(* CODESYS project MNG_SimIO_Upd.export

Project tree, tasks and I/O mapping:
  MNG_SimIO/
    function block MNG_SIMIO_UPDATER [ST]
  data type MNG_APPLICATION_INPUTS_32BIT
  data type MNG_APPLICATION_OUTPUTS_32BIT
*)

// MNG_APPLICATION_INPUTS_32BIT
TYPE MNG_APPLICATION_INPUTS_32BIT :
STRUCT
    NumSignals                    : INT     := 10        ;
EndoflEnd_of_Line_Packaging_STEP_TriggerZaehler_out: BOOL    := 0; (* EndoflEnd_of_Line_Packaging_STEP?TriggerZaehler_out *)

Gleitschiene_Links_AXIS: REAL    := 0.0; (* ubgeruest_EndoflGreifarm_Gleitschiene_Links?KinAxis *)

Laufwagen_1_Busy: BOOL    := 0; (* _EndoflEnd_of_Line_Packaging_STEP_Laufwagen_1?Busy *)

EndoflLaufwagen_AXIS: REAL    := 0.0; (* _Packaging_STEP_Laufwagen_1_EndoflLaufwagen?KinAxis *)

EndoflLaufwagen_DLT_POS: REAL    := 0.0; (* Packaging_STEP_Laufwagen_1_EndoflLaufwagen?KinDelta *)

EndoflLaufwagen_ACT_SPD: REAL    := 0.0; (* Packaging_STEP_Laufwagen_1_EndoflLaufwagen?KinSpeed *)

EndoflLaufwagen_KinState: DINT    := 0; (* Packaging_STEP_Laufwagen_1_EndoflLaufwagen?KinState *)

EndoflLaufwagen_ZaehlerQuer: UINT    := 0; (* kaging_STEP_Laufwagen_1_EndoflLaufwagen?ZaehlerQuer *)

EndoflLaufwagen_ZaehlerLaengs: UINT    := 0; (* ging_STEP_Laufwagen_1_EndoflLaufwagen?ZaehlerLaengs *)

EndoflLaufwagen_Hubausschiebpos: REAL    := 0.0; (* ng_STEP_Laufwagen_1_EndoflLaufwagen?Hubausschiebpos *)

END_STRUCT
END_TYPE

// MNG_APPLICATION_OUTPUTS_32BIT
TYPE MNG_APPLICATION_OUTPUTS_32BIT :
STRUCT
    NumSignals                    : INT     := 6         ;
Pusher_1_Enabled: BOOL    := 0; (* _EndoflEnd_of_Line_Packaging_STEP_Pusher_1?Enabled *)

Drehschieber_Achse_1_Set_AST: BOOL    := 0; (* ng_STEP_Drehschieber_1_Drehschieber_Achse_1?Set_AST *)

Drehschieber_Achse_1_Set_GST: BOOL    := 0; (* ng_STEP_Drehschieber_1_Drehschieber_Achse_1?Set_GST *)

EndoflEnd_of_Line_Packaging_STEP_Status_out: UINT    := 0; (* _EndoflEnd_of_Line_Packaging_STEP?Status_out *)

EndoflEnd_of_Line_Packaging_STEP_Ausschieben_in: BOOL    := 0; (* _EndoflEnd_of_Line_Packaging_STEP?Ausschieben_in *)

EndoflEnd_of_Line_Packaging_STEP_Laufwagen_1_Cmd_out: UINT    := 0; (* ndoflEnd_of_Line_Packaging_STEP?Laufwagen_1_Cmd_out *)

END_STRUCT
END_TYPE

// MNG_SimIO/MNG_SIMIO_UPDATER
FUNCTION_BLOCK MNG_SIMIO_UPDATER
(* This function block implements simple TCP/IP client protocol.              *)
(* The max. size of binary tx/rx data has to be <= PLCPRJ_BUFFER_SIZE         *)
VAR_INPUT
connect : BOOL := FALSE;
IPAddress : STRING := '192.168.8.175';
port : INT := 5003;
timeout : DINT := 3;		(* Timeout in seconds *)
Q : MNG_Application_Outputs_32Bit;    (* Tx user data *)
END_VAR
VAR_OUTPUT
I      : MNG_Application_Inputs_32Bit        ; (* Rx user data *)
Counter   : DINT := 0;
Connected : BOOL := FALSE;
END_VAR
VAR
state : INT := 0;
socket : RTS_IEC_HANDLE := -1(*SOCKET_INVALID*);
bOptNoDelay: BOOL := TRUE;
sa:SOCKADDRESS;
fdRead:SOCKET_FD_SET;
tvTimeout:SOCKET_TIMEVAL;
pdiReady:DINT := 0;
toServer         : MNG_RawDatagram;
fromServer       : MNG_RawDatagram;
expectedSize, recvSize : LINT := 0;
sendSize: UDINT := 0; 
sentSize : LINT := 0;

bInit: BOOL := FALSE;
DWordBuffer      : DWORD                                               ; (* convert DWORD data *)
DIntBuffer       : DINT                                                ; (* convert DINT data *)
Segment11_F: BOOL;
Error: DINT;
diSocket: BOOL;
result: RTS_IEC_RESULT; 
callback: CB.CB_CALLBACK;
callbackError: CB.ERROR; 
END_VAR
(* @END_DECLARATION := '0'                                                    *)

IF NOT bInit THEN
//         SysCallbackRegister(INDEXOF(CallbackReset), EVENT_BEFORE_RESET);
	callback.eEvent := CB.EVENT.BEFORE_RESET;
	callback.eClass := CB.EVENT_CLASS.ALL_CLASSES;
	callback.eSource := CB.EVENT_SOURCE.ALL_SOURCES;
	callback.pPOUFunc := ADR(CallbackReset); 
	
	CB.RegisterCallback(callback, ADR(callbackError));
        bInit := TRUE;
END_IF
CASE state OF
0:											(* Init *)
  	socket := -1(*SOCKET_INVALID*);
  	Connected := FALSE;
  	IF connect THEN
  	        state  := 10;
  	END_IF
10:											(* Create socket *)
        socket := SysSockCreate(SOCKET_AF_INET, SOCKET_STREAM, 0, ADR(result));
        (*IF socket <> 0(*= SOCKET_INVALID*) THEN
            state := 100;
        ELSE
            state := 20;
        END_IF*)
		state := 20;
20:											(* Setup and Connect *)
        (* SysSockSetOption(socket, SOCKET_SOL, SOCKET_SO_SNDBUF, ADR(diMaxDataSize), SIZEOF(diMaxDataSize));
        SysSockSetOption(socket, SOCKET_SOL, SOCKET_SO_RCVBUF, ADR(diMaxDataSize), SIZEOF(diMaxDataSize));
        lOptLinger.l_onoff:=0;
        lOptLinger.l_linger:=0;
        SysSockSetOption(diSocket,	SOCKET_SOL, SOCKET_SO_LINGER, ADR(lOptLinger), SIZEOF(lOptLinger)); *)
        bOptNoDelay:=TRUE;
        SysSockSetOption(socket,	SOCKET_IPPROTO_TCP, SOCKET_TCP_NODELAY, ADR(bOptNoDelay), SIZEOF(bOptNoDelay));
        sa.sin_family:=SOCKET_AF_INET;
        sa.sin_addr.ulAddr:=GetIPAddress(IPAddress);
        tvTimeout.tv_sec := timeout ;
        tvTimeout.tv_usec := 0;
        fdRead.fd_count := 1;
        fdRead.fd_array[0] := socket;
        IF sa.sin_addr.ulAddr = SOCKET_INADDR_NONE THEN
                state := 121;
        ELSE
                 sa.sin_port:=SysSockHtons(port);
                 IF SysSockConnect(socket, ADR(sa), SIZEOF(sa)) = 0  THEN
                        state := 30;
                 ELSE
                         Error := 10035(*SysSockGetLastErrorSync(socket)*);	
						(* Query reason why connect reported failure *)
                                         CASE  Error OF
                         10035: 			(* EWOULDBLOCK *)
                                 state := 30;
                         10056: 			 (* ALREADY_CONNECTED*)
                                 state := 30;
                         ELSE
                                 state := 60;
                         END_CASE
                END_IF
        END_IF
30:											(* Data exchange *)
                Connected := TRUE;
                fdRead.fd_array[0] := socket;
                IF (SysSockSelect(SOCKET_FD_SETSIZE, ADR(fdRead), 0, 0, ADR(tvTimeout), ADR(pdiReady)) = CmpErrors.Errors.ERR_OK) AND pdiReady > 0 THEN
                expectedSize := 16 + (I.NumSignals+1) * 4;
                recvSize := SysSockRecv(socket, ADR(fromServer), expectedSize, 0, ADR(result));
                IF result <> CmpErrors.Errors.ERR_OK OR expectedSize <= 0 THEN
                         state := 60;

                ELSIF expectedSize = recvSize THEN

                        (* correct header data *)
                        fromServer.Header.ByteCount   	 := SysSockNtohl(fromServer.Header.ByteCount);
                        Counter                        				:= SysSockNtohl(fromServer.Header.Counter);
                        fromServer.Header.SentTime  	   := SysSockNtohl(fromServer.Header.SentTime);
                        fromServer.Header.DatagramType := SysSockNtohl(fromServer.Header.DatagramType);

                        (* currently only use the data on a 32 Bit raw image *)
                        IF fromServer.Header.DatagramType = MNG_DatagramType.MNG_Raw32BitImage THEN
                                                        (* BOOL EndoflEnd_of_Line_Packaging_STEP_TriggerZaehler_out *)
                                                        I.EndoflEnd_of_Line_Packaging_STEP_TriggerZaehler_out := fromServer.Payload[2] <> 0;
                                                        (* REAL Gleitschiene_Links_AXIS *)
                                                        DWordBuffer := SysSockNtohl(fromServer.Payload[3]);
                                                        SysMemCpy(pDest := ADR(I.Gleitschiene_Links_AXIS), pSrc := ADR(DWordBuffer), udiCount := 4);
                                                        (* BOOL Laufwagen_1_Busy *)
                                                        I.Laufwagen_1_Busy := fromServer.Payload[4] <> 0;
                                                        (* REAL EndoflLaufwagen_AXIS *)
                                                        DWordBuffer := SysSockNtohl(fromServer.Payload[5]);
                                                        SysMemCpy(pDest := ADR(I.EndoflLaufwagen_AXIS), pSrc := ADR(DWordBuffer), udiCount := 4);
                                                        (* REAL EndoflLaufwagen_DLT_POS *)
                                                        DWordBuffer := SysSockNtohl(fromServer.Payload[6]);
                                                        SysMemCpy(pDest := ADR(I.EndoflLaufwagen_DLT_POS), pSrc := ADR(DWordBuffer), udiCount := 4);
                                                        (* REAL EndoflLaufwagen_ACT_SPD *)
                                                        DWordBuffer := SysSockNtohl(fromServer.Payload[7]);
                                                        SysMemCpy(pDest := ADR(I.EndoflLaufwagen_ACT_SPD), pSrc := ADR(DWordBuffer), udiCount := 4);
                                                        (* DINT EndoflLaufwagen_KinState *)
                                                        DWordBuffer := SysSockNtohl(fromServer.Payload[8]);
                                                        SysMemCpy(pDest := ADR(I.EndoflLaufwagen_KinState), pSrc := ADR(DWordBuffer), udiCount := 4);
                                                        (* UINT EndoflLaufwagen_ZaehlerQuer *)
                                                        DWordBuffer := SysSockNtohl(fromServer.Payload[9]);
                                                        I.EndoflLaufwagen_ZaehlerQuer := DWORD_TO_UINT(DWordBuffer);
                                                        (* UINT EndoflLaufwagen_ZaehlerLaengs *)
                                                        DWordBuffer := SysSockNtohl(fromServer.Payload[10]);
                                                        I.EndoflLaufwagen_ZaehlerLaengs := DWORD_TO_UINT(DWordBuffer);
                                                        (* REAL EndoflLaufwagen_Hubausschiebpos *)
                                                        DWordBuffer := SysSockNtohl(fromServer.Payload[11]);
                                                        SysMemCpy(pDest := ADR(I.EndoflLaufwagen_Hubausschiebpos), pSrc := ADR(DWordBuffer), udiCount := 4);
                                        state :=  40;
                END_IF
                END_IF
                ELSE
                state := 60;
                END_IF
40:											(* Send data *)
        sendSize := 16 + (Q.NumSignals+1) * 4;
        (*IF (SysSockSelect(SOCKET_FD_SETSIZE, ADR(fdRead), 0, 0, ADR(tvTimeout), ADR(result)) > 0) THEN*)
          toServer.Header.ByteCount    := SysSockHtonl(sendSize-16);
          toServer.Header.DatagramType := SysSockHtonl(MNG_DatagramType.MNG_Raw32BitImage);
          toServer.Header.Counter      := SysSockHtonl(Counter);
          toServer.Payload[1] := SysSockHtonl(Q.NumSignals); (* number of signals *)
                                                        (* BOOL Pusher_1_Enabled *)
                        IF Q.Pusher_1_Enabled = TRUE THEN
                            toServer.Payload[2] := 16#FFFFFFFF;   (*BOOL *)
                        ELSE
                            toServer.Payload[2] := 0;
                        END_IF;
                                                        (* BOOL Drehschieber_Achse_1_Set_AST *)
                        IF Q.Drehschieber_Achse_1_Set_AST = TRUE THEN
                            toServer.Payload[3] := 16#FFFFFFFF;   (*BOOL *)
                        ELSE
                            toServer.Payload[3] := 0;
                        END_IF;
                                                        (* BOOL Drehschieber_Achse_1_Set_GST *)
                        IF Q.Drehschieber_Achse_1_Set_GST = TRUE THEN
                            toServer.Payload[4] := 16#FFFFFFFF;   (*BOOL *)
                        ELSE
                            toServer.Payload[4] := 0;
                        END_IF;
                                                        (* UINT EndoflEnd_of_Line_Packaging_STEP_Status_out *)
                        DWordBuffer := UINT_TO_DWORD(Q.EndoflEnd_of_Line_Packaging_STEP_Status_out);
                        toServer.Payload[5] := SysSockHtonl(DWordBuffer);
                                                        (* BOOL EndoflEnd_of_Line_Packaging_STEP_Ausschieben_in *)
                        IF Q.EndoflEnd_of_Line_Packaging_STEP_Ausschieben_in = TRUE THEN
                            toServer.Payload[6] := 16#FFFFFFFF;   (*BOOL *)
                        ELSE
                            toServer.Payload[6] := 0;
                        END_IF;
                                                        (* UINT EndoflEnd_of_Line_Packaging_STEP_Laufwagen_1_Cmd_out *)
                        DWordBuffer := UINT_TO_DWORD(Q.EndoflEnd_of_Line_Packaging_STEP_Laufwagen_1_Cmd_out);
                        toServer.Payload[7] := SysSockHtonl(DWordBuffer);
        (*    toServer.Header.SentTime := SysSockHtonl(clock.systemTime.wMilliseconds + clock.systemTime.wMinute * 60000); *)
            sentSize := SysSockSend(socket, ADR(toServer), sendSize, 0, ADR(result));
            IF sentSize < 0 THEN
               state := 60;
            ELSE
               state := 30;
            END_IF
        (*ELSE
                        state := 60;
        END_IF*)
60:											(* Disconnect *)
                IF socket = 0(*SOCKET_INVALID*) THEN
                                state := 0;
                ELSE
                                IF SysSockClose(socket) <> 0(*= FALSE*) THEN
                                          state := 161;
                                ELSE
                                                state := 70;
                                END_IF
          END_IF
70:											(* Delete socket *)
          IF socket = 0(*SOCKET_INVALID*) THEN
                                state := 0;
                ELSE
                    IF SysSockShutdown(socket, 0) <> 0(*= FALSE*) THEN
                                          state := 0;
                                ELSE
                                                state := 0;
                                END_IF
          END_IF
110:										(* Error Create socket failed *)
;
121:										(* Error IP number invalid *)
;
122:										(* Error connect failed *)
     state := 70;
131:										(* Error while receiving, received bytes < expected)*)
                 state := 60;
161: 										(* Error close failed *)
;
END_CASE
IF NOT connect AND state> 0 AND state < 60 THEN
                state := 60;
END_IF

END_FUNCTION_BLOCK
